// Mitsubishi GX Works2 project: Industrial Automation CA2   PLC: FX2N/FX2NC

PROGRAM MAIN
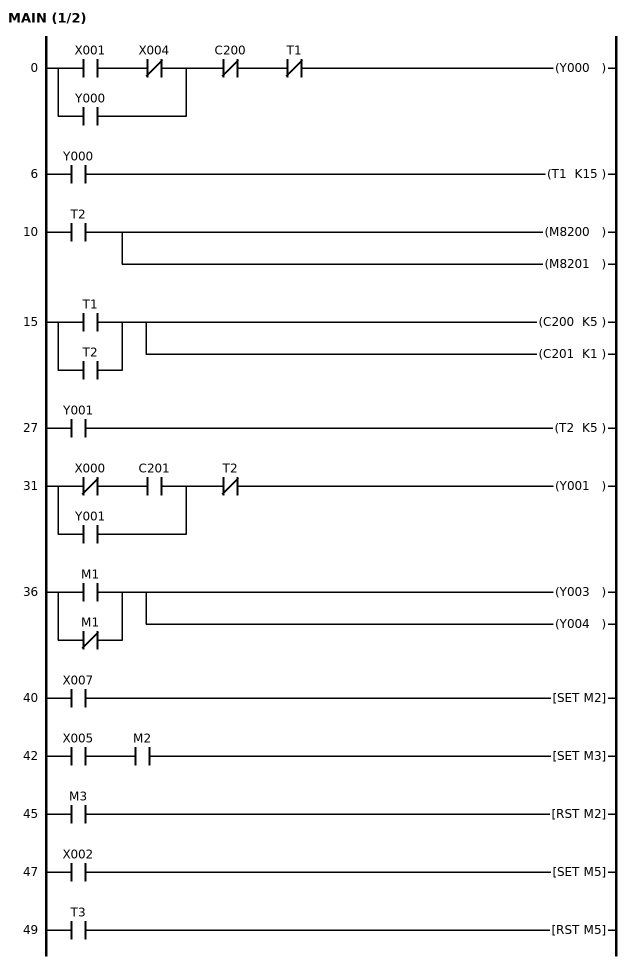
0     LD      X001
      ANI     X004
      OR      Y000
      ANI     C200
      ANI     T1
      OUT     Y000
6     LD      Y000
      OUT     T1 K15
10    LD      T2
      OUT     M8200
      OUT     M8201
15    LD      T1
      OR      T2
      OUT     C200 K5
      OUT     C201 K1
27    LD      Y001
      OUT     T2 K5
31    LDI     X000
      AND     C201
      OR      Y001
      ANI     T2
      OUT     Y001
36    LD      M1
      ORI     M1
      OUT     Y003
      OUT     Y004
40    LD      X007
      SET     M2
42    LD      X005
      AND     M2
      SET     M3
45    LD      M3
      RST     M2
47    LD      X002
      SET     M5
49    LD      T3
      RST     M5
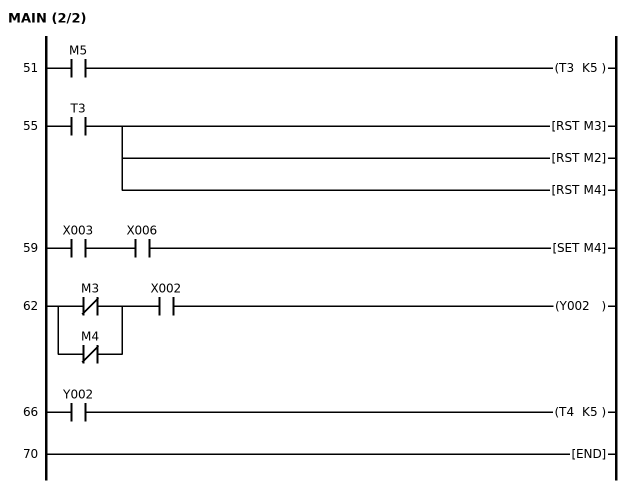
51    LD      M5
      OUT     T3 K5
55    LD      T3
      RST     M3
      RST     M2
      RST     M4
59    LD      X003
      AND     X006
      SET     M4
62    LDI     M3
      ORI     M4
      AND     X002
      OUT     Y002
66    LD      Y002
      OUT     T4 K5
70    END
END_PROGRAM
